// Mitsubishi GX Works2 project: semaforo1   PLC: Q03UDV

PROGRAM MAIN
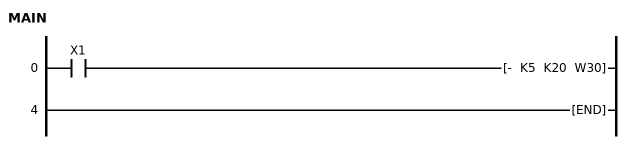
0     LD      X1
      -       K5 K20 W30
4     END
END_PROGRAM
